PROGRAM P800_Core_Messaging
VAR
END_VAR

// if flag goes high from service set it low and bump counter
IF (vMessages.SQL_ExceptionFlag > 0) THEN
	vMessages.SQL_ExceptionFlag :=0;
	vMessages.SQL_ExceptionCount := SQL_ExceptionCount + 1;	
	// cap exception count
	IF (vMessages.SQL_ExceptionCount > 10001 )THEN
		vMessages.SQL_ExceptionCount := 10001;
	END_IF	
END_IF


IF SCP.DisableMessaging THEN
	RETURN;
END_IF

// Process whatever buffers you want here
sMsg_Process_Buffer(Msgs_SCP);      // generic SCP message buffer
sMsg_Process_Buffer(Msgs_Itm);      // Itmsort SCP message buffer
sMsg_Process_Buffer(Msgs_Ind);      // Itmsort FAST SCP message buffer
sMsg_Process_Buffer(Msgs_Log);      // Multithreaded, used for silent messages/heartbeat

END_PROGRAM

(* stored: Version 1.1.0.1, ProductVersion 3.1.4024.9
   POU P800_Core_Messaging: Id {ae625f7e-0929-4f56-bdd1-e329f26ca566}, SpecialFunc None *)
